{attribute 'linkalways'} 
{attribute 'no_explicit_call' := 'This FB is a CLASS and must be accessed using methods or properties'}
{attribute 'enable_dynamic_creation'}
FUNCTION_BLOCK Node_F_VN_Histogram EXTENDS VisionNode
VAR
	ipSrcImage : _ITcVnImage;
    ipDestHistogram : _ITcVnContainer;
    hrPrev : _HRESULT(S_OK);
	hresult : _HRESULT(S_OK);
END_VAR

METHOD PUBLIC  Clone : I_Node
VAR
	pNode : POINTER TO Node_F_VN_Histogram;
END_VAR
pNode := __NEW(Node_F_VN_Histogram);
Clone := pNode^;
END_METHOD

METHOD FB_init : BOOL
VAR_INPUT
	bInitRetains : BOOL; // if TRUE, the retain variables are initialized (warm start / cold start)
	bInCopyCode : BOOL;  // if TRUE, the instance afterwards gets moved into the copy code (online change)
END_VAR
AddInput('ipSrcImage', ipSrcImage);
AddInput('hrPrev', hrPrev);
AddOutput('ipDestHistogram', ipDestHistogram);
AddOutput('hresult',hresult);
END_METHOD

METHOD PROTECTED  OnExecute : HRESULT
hresult.Value := F_VN_Histogram(
	ipSrcImage := ipSrcImage.Value,
    ipDestHistogram := ipDestHistogram.Value,
	hrPrev := hrPrev.Value);
END_METHOD

METHOD PUBLIC PreExecutionCheck
VAR_INPUT
	Check : I_PreExecutionChecks;
END_VAR
VAR
    colorMapSize : ULINT;
END_VAR
Check.IsTrue(ipSrcImage.IsValid, 'ipSrcImage must contain an image');
END_METHOD

END_FUNCTION_BLOCK

(* stored: Version 1.1.0.1, ProductVersion 3.1.4024.13
   POU Node_F_VN_Histogram: Id {b97d7b4f-b4b8-02ec-07a6-6d42e09ad70c}, SpecialFunc None
   Folder Constructor: Id {2b5a5459-bc39-0b5b-3fec-1e89872db5a4}
   Method Clone: Id {b9d0b98f-266f-0aa4-3394-9441f8cb962a}
   Method FB_init: Id {db72bb6b-a7b7-020f-3166-19d74fa8fd20}
   Method OnExecute: Id {7b2d6f65-c174-0f29-1035-281da0501c8b}
   Method PreExecutionCheck: Id {192c8930-758e-0b66-1d84-d76292c2b35e} *)
